SUBAPPLICATION SystemTick (* Freilaufender Tick-Zaehler (0..99, alle 200ms +1) als ADI-Ausgang - Lebenszeichen/Heartbeat *)
  (* Standard: 61499-2; Description: Copyright (c) 2026 Meisterschulen am Ostbahnhof This program and the accompanying materials are made available under the terms of the Eclipse Public License 2.0 which is available at https://www.eclipse.org/legal/epl-2.0/ SPDX-License-Identifier: EPL-2.0 *)
  (* Version 1.0, 2026-08-07, Franz Höpfinger, Meisterschulen am Ostbahnhof, initial API and implementation and/or initial documentation *)
  PACKAGE MyLib::sys;
  (* Documentation:
  Freilaufender Tick-Zähler (Heartbeat)
   Zählt ohne externen Trigger alle 200ms um 1 hoch und läuft bei 100 wieder auf 0 zurück (Zyklus = 20s). Der aktuelle Zählerstand wird als ADI_OUT (1 Event + 1 DINT) bereitgestellt. Dient als Lebenszeichen: solange sich der Wert weiter ändert, läuft die Steuerung, die ihn erzeugt, noch - egal ob er lokal auf dem VT angezeigt (SystemTickSender_ISO) oder per OPC-UA an ein anderes Modul verteilt wird (SystemTickSender_OPC).
   Funktionsbeschreibung
    - INIT startet einmalig E_CYCLE (Periode 200ms über DT).
   - Jeder Zyklus erhöht den intern über F_MOVE/ADD_2 gehaltenen Zähler um 1 (IN1=DINT#1).
   - F_MOD (Modulo 100) begrenzt den sichtbaren Wert auf den Bereich 0..99.
   - ADI_DINT_TO_DI verpackt den DINT-Wert in das ADI-Adapterformat für den Plug ADI_OUT.
  *)
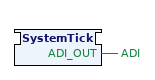
  PLUGS
    ADI_OUT : adapter::types::unidirectional::ADI; (* Aktueller Tick-Zaehlerstand (0..99), aendert sich alle 200ms *)
  END_PLUGS
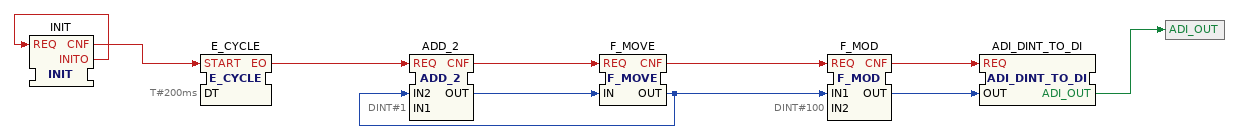
  FBS
    F_MOD : iec61131::arithmetic::F_MOD(IN2 := DINT#100);
    ADD_2 : iec61131::arithmetic::ADD_2(IN1 := DINT#1);
    E_CYCLE : iec61499::events::E_CYCLE(DT := T#200ms);
    INIT : iec61131::booleanOperators::INIT;
    F_MOVE : iec61131::selection::F_MOVE; {SET_ATTRIBUTE(DataType, DINT)}
    ADI_DINT_TO_DI : adapter::conversion::unidirectional::ADI_DINT_TO_DI;
  END_FBS
  EVENT_CONNECTIONS
    F_MOVE.CNF TO F_MOD.REQ;
    F_MOD.CNF TO ADI_DINT_TO_DI.REQ;
    E_CYCLE.EO TO ADD_2.REQ;
    ADD_2.CNF TO F_MOVE.REQ;
    INIT.CNF TO E_CYCLE.START;
    INIT.INITO TO INIT.REQ;
  END_CONNECTIONS
  DATA_CONNECTIONS
    F_MOVE.OUT TO F_MOD.IN1;
    F_MOD.OUT TO ADI_DINT_TO_DI.OUT;
    F_MOVE.OUT TO ADD_2.IN2;
    ADD_2.OUT TO F_MOVE.IN;
  END_CONNECTIONS
  ADAPTER_CONNECTIONS
    ADI_DINT_TO_DI.ADI_OUT TO ADI_OUT;
  END_CONNECTIONS
END_SUBAPPLICATION
